// TIA Portal project "Magazzino" (V17)
// Vorlageprojekt für das Buch mit Zielsystem S7-1200

(* hardware
DEVICE "S7-1200-Station_1"  S7-1200 Station
   slot 0: "Baugruppenträger_0"  Rack  V1.0
   slot 1: "PLC_1"  CPU 1211C DC/DC/DC  6ES7 211-1AE40-0XB0  V4.1
DEVICE "HMI_1"  KTP900 Basic PN
   slot 0: "HMI_1"  KTP900 Basic PN  6AV2 123-2JB03-0AX0  17.0.0.0
   slot 1: "HMI_RT_2"  KTP900 Basic PN  6AV2 123-2JB03-0AX0  17.0.0.0
   slot 5: "HMI_1.IE_CP_1"  PROFINET Interface  17.0.0.0
      slot 1: "PROFINET Interface_1"  PROFINET Interface
         slot 1: "Port_1"  Port
*)

// ===== PLC "PLC_1"  CPU 1211C DC/DC/DC =====

VAR_GLOBAL   // PLC tag table "nastro_pacchi"
   "PaccoSens" AT %I0.0 : Bool;
   "Motor_pacchi" AT %Q0.0 : Bool;
END_VAR

VAR_GLOBAL   // PLC tag table "nastro_pedana"
   "PedanaSens" AT %I0.1 : Bool;
   "Motor_pedane" AT %Q0.1 : Bool;
END_VAR

VAR_GLOBAL   // PLC tag table "nastro_uscita"
   "FineSens" AT %I0.2 : Bool;
   "Motor" AT %Q0.2 : Bool;
END_VAR

VAR_GLOBAL   // PLC tag table "robot"
   "GoDownSens" AT %I0.3 : Bool;
   "GrabSens" AT %I0.4 : Bool;
   "MoveSens" AT %I0.5 : Bool;
   "GoDown" AT %Q0.3 : Bool;
   "Grab" AT %Q0.4 : Bool;
   "Move" AT %Q0.5 : Bool;
END_VAR

VAR_GLOBAL   // PLC tag table "allineatore"
   "AllineaSens" AT %I0.6 : Bool;
   "Allinea" AT %Q0.6 : Bool;
END_VAR

VAR_GLOBAL   // PLC tag table "bilancia"
   "BilanciaSens" AT %I1.2 : Bool;
   "Motor_bilancia" AT %Q1.1 : Bool;
   "BilanciaPeso" AT %ID30 : Real;
END_VAR

VAR_GLOBAL   // PLC tag table "stacker"
   "CentroSens" AT %I1.3 : Bool;
   "StackerMoveSens" AT %I1.4 : Bool;
   "PrelevaRSens" AT %I1.5 : Bool;
   "PrelevaLSens" AT %I1.6 : Bool;
   "AlzaSens" AT %I1.7 : Bool;
   "PrelevaR" AT %Q1.2 : Bool;
   "PrelevaL" AT %Q1.3 : Bool;
   "Alza" AT %Q1.4 : Bool;
   "Posizione" AT %QD30 : DInt;
END_VAR

VAR_GLOBAL   // PLC tag table "loader_carica"
   "CaricaSens" AT %I1.0 : Bool;
   "PaccoSuPallet" AT %I0.7 : Bool;
   "Carica" AT %Q0.7 : Bool;
END_VAR

VAR_GLOBAL   // PLC tag table "loader_scarica"
   "ScaricaSens" AT %I1.1 : Bool;
   "Scarica" AT %Q1.0 : Bool;
END_VAR

DATA_BLOCK "Database"   // DB1
{ S7_Optimized_Access := 'TRUE' }
VERSION : 0.1
   VAR
      "Mod" : Bool := true;
      Peso : Real;
      Posizione : DInt;
      CodaPesi : Array[0..4] of Real;
      HeadPesi : Int;
      TailPesi : Int;
      ArrayMagazzino : Array[0..54] of Bool;
      PosLibere : Int := 54;
   END_VAR
BEGIN
END_DATA_BLOCK

DATA_BLOCK "Magazzino_DB"   // DB2
{ S7_Optimized_Access := 'TRUE' }
VERSION : 0.1
// stored: InstanceOfName Magazzino
"Magazzino"
BEGIN
END_DATA_BLOCK

FUNCTION_BLOCK "Bilancia"   // FB1, LAD
{ S7_Optimized_Access := 'TRUE' }
VERSION : 0.1
   VAR_INPUT
      BilanciaSens : Bool;
      BilanciaPeso : Real;
      allineatore_ok : Bool;
      robot_ok : Bool;
   END_VAR
   VAR_OUTPUT
      motor_bilancia : Bool;
      p_acc : Bool;
      allineatore_start : Bool;
      robot_start : Bool;
   END_VAR
   VAR
      INIT : Bool;
      F0 : Bool;
      F1 : Bool;
      F2 : Bool;
      F3 : Bool;
      TR0 : Bool;
      TR1 : Bool;
      TR2 : Bool;
      TR3 : Bool;
      timer1 : TON_TIME;
      timer2 : TON_TIME;
      R_BilanciaSens : R_TRIG;
      F_BilanciaSens : F_TRIG;
      R_allineatore_ok : R_TRIG;
      R_F2 : R_TRIG;
      R_Inserisci : R_TRIG;
      R_robot_ok : R_TRIG;
      Inserisci : Bool;
      Salva : Bool;
   END_VAR
   VAR_TEMP   // added for the SCL form of the ladder/FBD networks
      _w1 : Bool;
   END_VAR
BEGIN

REGION Network 1: INIZIALIZZAZIONE
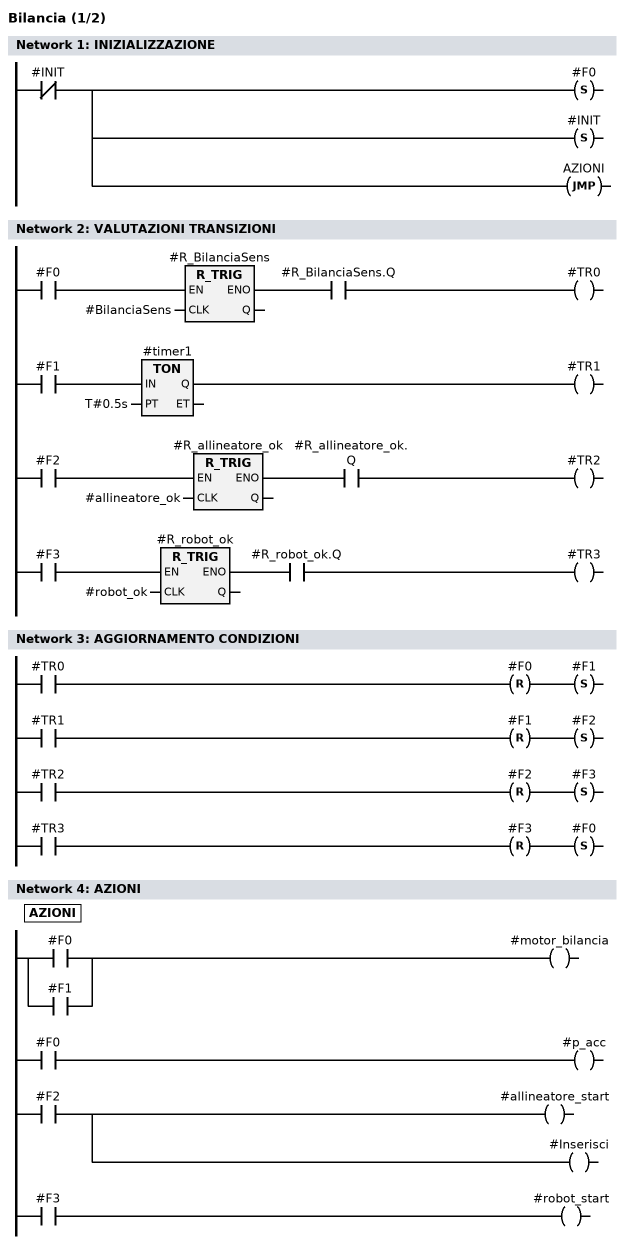
   RUNG wire#powerrail
      I_Contact( #INIT )
      wire#w1
      S_Coil( #F0 )
   END_RUNG
   RUNG wire#w1
      S_Coil( #INIT )
   END_RUNG
   RUNG wire#w1
      JumpCoil( AZIONI )
   END_RUNG
   // the same network as SCL:
   IF NOT #INIT THEN #F0 := TRUE; END_IF;
   #_w1 := NOT #INIT;
   IF #_w1 THEN
       #INIT := TRUE;
       GOTO AZIONI;
   END_IF;
END_REGION

REGION Network 2: VALUTAZIONI TRANSIZIONI
   // ENO of a box is taken as its EN; it also drops when the box reports an error
   IF #F0 THEN
       #R_BilanciaSens(CLK := #BilanciaSens);   // R_TRIG
   END_IF;
   #TR0 := #F0 AND #R_BilanciaSens.Q;
   #timer1(IN := #F1, PT := T#0.5s);   // TON
   #TR1 := #timer1.Q;
   IF #F2 THEN
       #R_allineatore_ok(CLK := #allineatore_ok);   // R_TRIG
   END_IF;
   #TR2 := #F2 AND #R_allineatore_ok.Q;
   IF #F3 THEN
       #R_robot_ok(CLK := #robot_ok);   // R_TRIG
   END_IF;
   #TR3 := #F3 AND #R_robot_ok.Q;
END_REGION

REGION Network 3: AGGIORNAMENTO CONDIZIONI
   RUNG wire#powerrail
      Contact( #TR0 )
      R_Coil( #F0 )
      S_Coil( #F1 )
   END_RUNG
   RUNG wire#powerrail
      Contact( #TR1 )
      R_Coil( #F1 )
      S_Coil( #F2 )
   END_RUNG
   RUNG wire#powerrail
      Contact( #TR2 )
      R_Coil( #F2 )
      S_Coil( #F3 )
   END_RUNG
   RUNG wire#powerrail
      Contact( #TR3 )
      R_Coil( #F3 )
      S_Coil( #F0 )
   END_RUNG
   // the same network as SCL:
   IF #TR0 THEN
       #F0 := FALSE;
       #F1 := TRUE;
   END_IF;
   IF #TR1 THEN
       #F1 := FALSE;
       #F2 := TRUE;
   END_IF;
   IF #TR2 THEN
       #F2 := FALSE;
       #F3 := TRUE;
   END_IF;
   IF #TR3 THEN
       #F3 := FALSE;
       #F0 := TRUE;
   END_IF;
END_REGION

REGION Network 4: AZIONI
   Label( AZIONI )
   RUNG wire#powerrail
      Contact( #F0 )
      wire#w1
      Coil( #motor_bilancia )
   END_RUNG
   RUNG wire#powerrail
      Contact( #F1 )
   END_RUNG wire#w1
   RUNG wire#powerrail
      Contact( #F0 )
      Coil( #p_acc )
   END_RUNG
   RUNG wire#powerrail
      Contact( #F2 )
      wire#w2
      Coil( #allineatore_start )
   END_RUNG
   RUNG wire#w2
      Coil( #Inserisci )
   END_RUNG
   RUNG wire#powerrail
      Contact( #F3 )
      Coil( #robot_start )
   END_RUNG
   // the same network as SCL:
   AZIONI:
   #motor_bilancia := #F0 OR #F1;
   #p_acc := #F0;
   #allineatore_start := #F2;
   #Inserisci := #F2;
   #robot_start := #F3;
END_REGION

REGION Network 5: GESTIONE CODA PESI
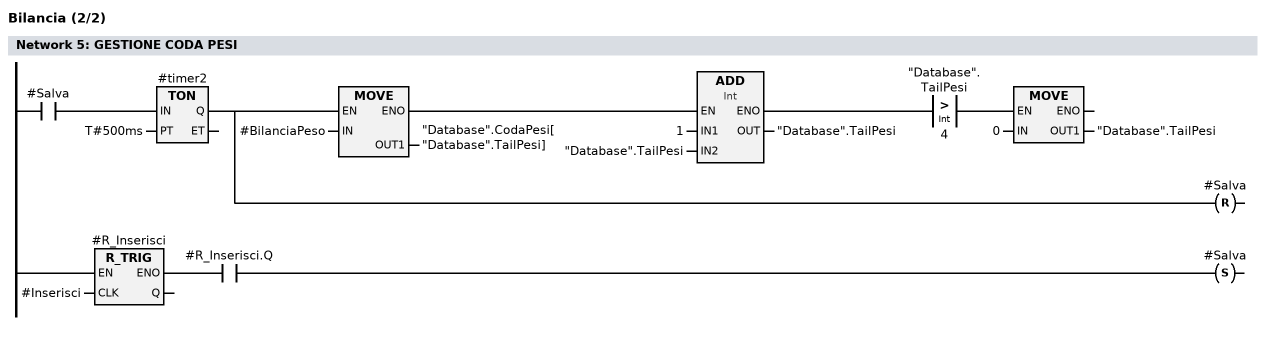
   // ENO of a box is taken as its EN; it also drops when the box reports an error
   #timer2(IN := #Salva, PT := T#500ms);   // TON
   IF #timer2.Q THEN
       "Database".CodaPesi["Database".TailPesi] := #BilanciaPeso;
       "Database".TailPesi := 1 + "Database".TailPesi;
   END_IF;
   IF #timer2.Q AND ("Database".TailPesi > 4) THEN "Database".TailPesi := 0; END_IF;
   IF #timer2.Q THEN #Salva := FALSE; END_IF;
   #R_Inserisci(CLK := #Inserisci);   // R_TRIG
   IF #R_Inserisci.Q THEN #Salva := TRUE; END_IF;
END_REGION
END_FUNCTION_BLOCK

FUNCTION_BLOCK "Robot"   // FB2, LAD
{ S7_Optimized_Access := 'TRUE' }
VERSION : 0.1
   VAR_INPUT
      MoveSens : Bool;
      GrabSens : Bool;
      GoDownSens : Bool;
      start : Bool;
      loader_ok : Bool;
   END_VAR
   VAR_OUTPUT
      Move : Bool;
      Grab : Bool;
      GoDown : Bool;
      fine : Bool;
      pacco_pronto : Bool;
   END_VAR
   VAR
      f0 : Bool;
      f1 : Bool;
      f2 : Bool;
      f3 : Bool;
      f4 : Bool;
      f5 : Bool;
      f6 : Bool;
      f7 : Bool;
      f8 : Bool;
      TR0 : Bool;
      TR1 : Bool;
      TR2 : Bool;
      TR3 : Bool;
      TR5 : Bool;
      TR6 : Bool;
      TR7 : Bool;
      TR8 : Bool;
      INIZ : Bool;
      r_prendi : R_TRIG;
      r_GrabSens : R_TRIG;
      f_GoDownSens : F_TRIG;
      f_MoveSens : F_TRIG;
      timer1 : TON_TIME;
   END_VAR
   VAR_TEMP   // added for the SCL form of the ladder/FBD networks
      _w1 : Bool;
   END_VAR
BEGIN

REGION Network 1: Inizializzazione
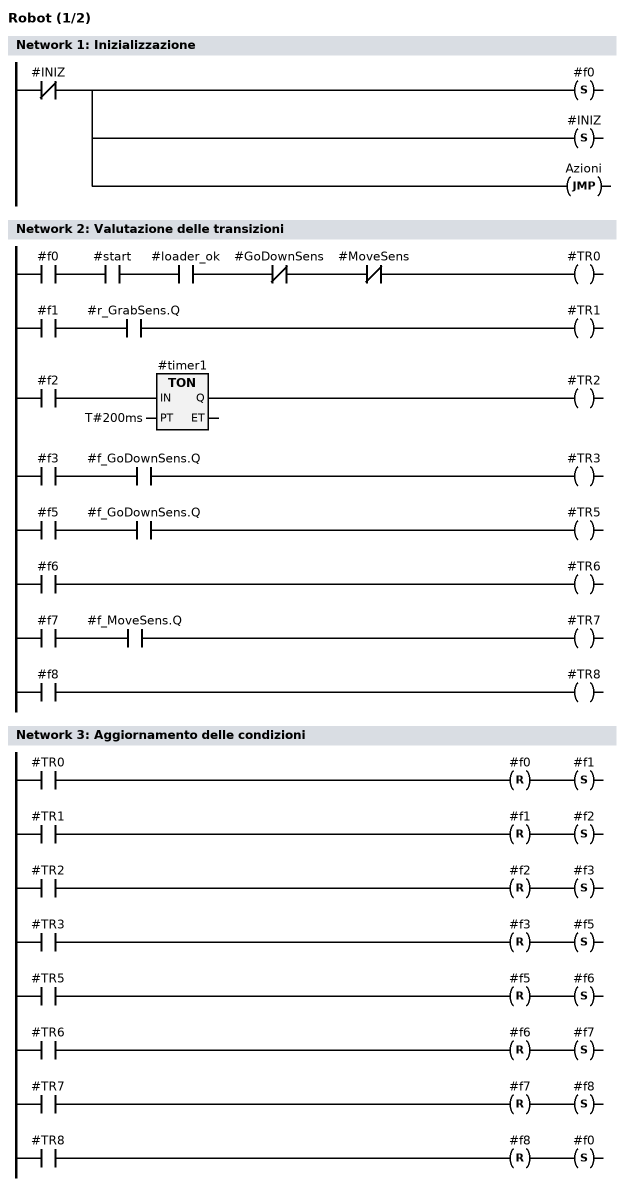
   RUNG wire#powerrail
      I_Contact( #INIZ )
      wire#w1
      S_Coil( #f0 )
   END_RUNG
   RUNG wire#w1
      S_Coil( #INIZ )
   END_RUNG
   RUNG wire#w1
      JumpCoil( Azioni )
   END_RUNG
   // the same network as SCL:
   IF NOT #INIZ THEN #f0 := TRUE; END_IF;
   #_w1 := NOT #INIZ;
   IF #_w1 THEN
       #INIZ := TRUE;
       GOTO Azioni;
   END_IF;
END_REGION

REGION Network 2: Valutazione delle transizioni
   #TR0 := #f0 AND #start AND #loader_ok AND NOT #GoDownSens AND NOT #MoveSens;
   #TR1 := #f1 AND #r_GrabSens.Q;
   #timer1(IN := #f2, PT := T#200ms);   // TON
   #TR2 := #timer1.Q;
   #TR3 := #f3 AND #f_GoDownSens.Q;
   #TR5 := #f5 AND #f_GoDownSens.Q;
   #TR6 := #f6;
   #TR7 := #f7 AND #f_MoveSens.Q;
   #TR8 := #f8;
END_REGION

REGION Network 3: Aggiornamento delle condizioni
   RUNG wire#powerrail
      Contact( #TR0 )
      R_Coil( #f0 )
      S_Coil( #f1 )
   END_RUNG
   RUNG wire#powerrail
      Contact( #TR1 )
      R_Coil( #f1 )
      S_Coil( #f2 )
   END_RUNG
   RUNG wire#powerrail
      Contact( #TR2 )
      R_Coil( #f2 )
      S_Coil( #f3 )
   END_RUNG
   RUNG wire#powerrail
      Contact( #TR3 )
      R_Coil( #f3 )
      S_Coil( #f5 )
   END_RUNG
   RUNG wire#powerrail
      Contact( #TR5 )
      R_Coil( #f5 )
      S_Coil( #f6 )
   END_RUNG
   RUNG wire#powerrail
      Contact( #TR6 )
      R_Coil( #f6 )
      S_Coil( #f7 )
   END_RUNG
   RUNG wire#powerrail
      Contact( #TR7 )
      R_Coil( #f7 )
      S_Coil( #f8 )
   END_RUNG
   RUNG wire#powerrail
      Contact( #TR8 )
      R_Coil( #f8 )
      S_Coil( #f0 )
   END_RUNG
   // the same network as SCL:
   IF #TR0 THEN
       #f0 := FALSE;
       #f1 := TRUE;
   END_IF;
   IF #TR1 THEN
       #f1 := FALSE;
       #f2 := TRUE;
   END_IF;
   IF #TR2 THEN
       #f2 := FALSE;
       #f3 := TRUE;
   END_IF;
   IF #TR3 THEN
       #f3 := FALSE;
       #f5 := TRUE;
   END_IF;
   IF #TR5 THEN
       #f5 := FALSE;
       #f6 := TRUE;
   END_IF;
   IF #TR6 THEN
       #f6 := FALSE;
       #f7 := TRUE;
   END_IF;
   IF #TR7 THEN
       #f7 := FALSE;
       #f8 := TRUE;
   END_IF;
   IF #TR8 THEN
       #f8 := FALSE;
       #f0 := TRUE;
   END_IF;
END_REGION

REGION Network 4: Azioni
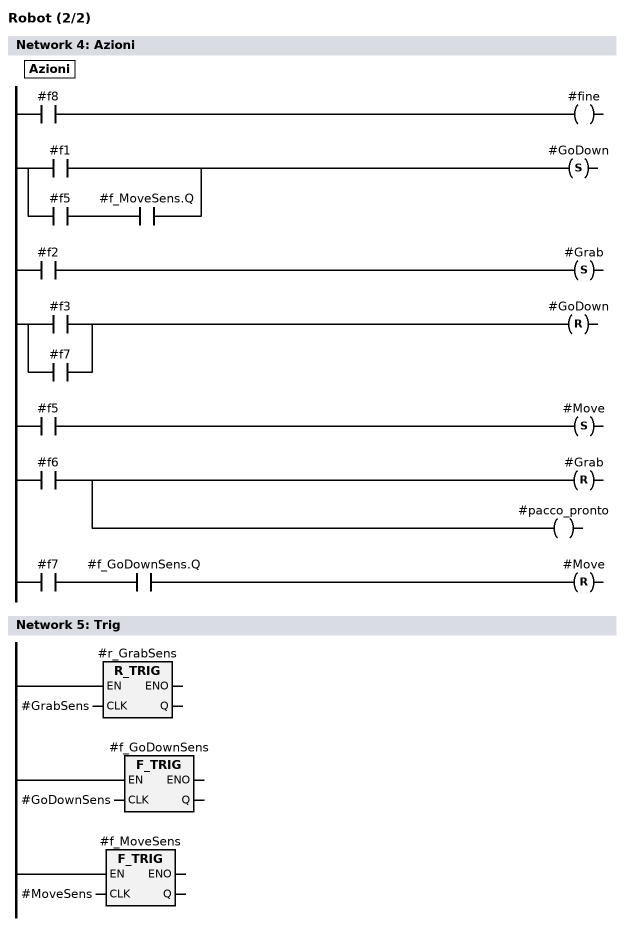
   Label( Azioni )
   RUNG wire#powerrail
      Contact( #f8 )
      Coil( #fine )
   END_RUNG
   RUNG wire#powerrail
      Contact( #f1 )
      wire#w1
      S_Coil( #GoDown )
   END_RUNG
   RUNG wire#powerrail
      Contact( #f5 )
      Contact( #f_MoveSens.Q )
   END_RUNG wire#w1
   RUNG wire#powerrail
      Contact( #f2 )
      S_Coil( #Grab )
   END_RUNG
   RUNG wire#powerrail
      Contact( #f3 )
      wire#w2
      R_Coil( #GoDown )
   END_RUNG
   RUNG wire#powerrail
      Contact( #f7 )
   END_RUNG wire#w2
   RUNG wire#powerrail
      Contact( #f5 )
      S_Coil( #Move )
   END_RUNG
   RUNG wire#powerrail
      Contact( #f6 )
      wire#w3
      R_Coil( #Grab )
   END_RUNG
   RUNG wire#w3
      Coil( #pacco_pronto )
   END_RUNG
   RUNG wire#powerrail
      Contact( #f7 )
      Contact( #f_GoDownSens.Q )
      R_Coil( #Move )
   END_RUNG
   // the same network as SCL:
   Azioni:
   #fine := #f8;
   IF #f1 OR (#f5 AND #f_MoveSens.Q) THEN #GoDown := TRUE; END_IF;
   IF #f2 THEN #Grab := TRUE; END_IF;
   IF #f3 OR #f7 THEN #GoDown := FALSE; END_IF;
   IF #f5 THEN #Move := TRUE; END_IF;
   IF #f6 THEN #Grab := FALSE; END_IF;
   #pacco_pronto := #f6;
   IF #f7 AND #f_GoDownSens.Q THEN #Move := FALSE; END_IF;
END_REGION

REGION Network 5: Trig
   #r_GrabSens(CLK := #GrabSens);   // R_TRIG
   #f_GoDownSens(CLK := #GoDownSens);   // F_TRIG
   #f_MoveSens(CLK := #MoveSens);   // F_TRIG
END_REGION
END_FUNCTION_BLOCK

FUNCTION_BLOCK "Loader"   // FB3, LAD
{ S7_Optimized_Access := 'TRUE' }
VERSION : 0.1
   VAR_INPUT
      s : Bool;
      p_dopo : Bool;
      pacco : Bool;
      flag : Bool;
   END_VAR
   VAR_OUTPUT
      motor : Bool;
      p_acc : Bool;
      posa : Bool;
      p_cons : Bool;
   END_VAR
   VAR
      INIT : Bool;
      F0 : Bool;
      F1 : Bool;
      F01 : Bool;
      F11 : Bool;
      TR0 : Bool;
      TR1 : Bool;
      TR2 : Bool;
      TR3 : Bool;
      TR4 : Bool;
      F_S : F_TRIG;
      R_S : R_TRIG;
      R_pacco : R_TRIG;
   END_VAR
   VAR_TEMP   // added for the SCL form of the ladder/FBD networks
      _w1 : Bool;
   END_VAR
BEGIN

REGION Network 1: INIZIALIZZAZIONE
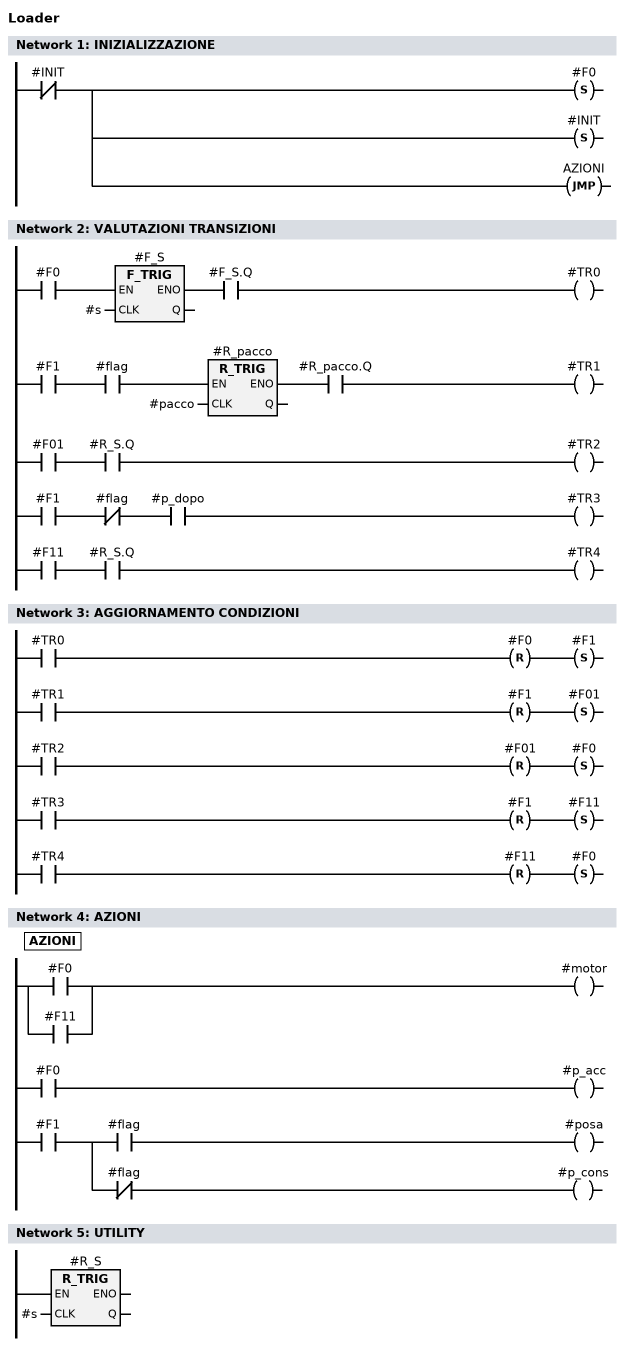
   RUNG wire#powerrail
      I_Contact( #INIT )
      wire#w1
      S_Coil( #F0 )
   END_RUNG
   RUNG wire#w1
      S_Coil( #INIT )
   END_RUNG
   RUNG wire#w1
      JumpCoil( AZIONI )
   END_RUNG
   // the same network as SCL:
   IF NOT #INIT THEN #F0 := TRUE; END_IF;
   #_w1 := NOT #INIT;
   IF #_w1 THEN
       #INIT := TRUE;
       GOTO AZIONI;
   END_IF;
END_REGION

REGION Network 2: VALUTAZIONI TRANSIZIONI
   // ENO of a box is taken as its EN; it also drops when the box reports an error
   IF #F0 THEN
       #F_S(CLK := #s);   // F_TRIG
   END_IF;
   #TR0 := #F0 AND #F_S.Q;
   #_w1 := #F1 AND #flag;
   IF #_w1 THEN
       #R_pacco(CLK := #pacco);   // R_TRIG
   END_IF;
   #TR1 := #_w1 AND #R_pacco.Q;
   #TR2 := #F01 AND #R_S.Q;
   #TR3 := #F1 AND NOT #flag AND #p_dopo;
   #TR4 := #F11 AND #R_S.Q;
END_REGION

REGION Network 3: AGGIORNAMENTO CONDIZIONI
   RUNG wire#powerrail
      Contact( #TR0 )
      R_Coil( #F0 )
      S_Coil( #F1 )
   END_RUNG
   RUNG wire#powerrail
      Contact( #TR1 )
      R_Coil( #F1 )
      S_Coil( #F01 )
   END_RUNG
   RUNG wire#powerrail
      Contact( #TR2 )
      R_Coil( #F01 )
      S_Coil( #F0 )
   END_RUNG
   RUNG wire#powerrail
      Contact( #TR3 )
      R_Coil( #F1 )
      S_Coil( #F11 )
   END_RUNG
   RUNG wire#powerrail
      Contact( #TR4 )
      R_Coil( #F11 )
      S_Coil( #F0 )
   END_RUNG
   // the same network as SCL:
   IF #TR0 THEN
       #F0 := FALSE;
       #F1 := TRUE;
   END_IF;
   IF #TR1 THEN
       #F1 := FALSE;
       #F01 := TRUE;
   END_IF;
   IF #TR2 THEN
       #F01 := FALSE;
       #F0 := TRUE;
   END_IF;
   IF #TR3 THEN
       #F1 := FALSE;
       #F11 := TRUE;
   END_IF;
   IF #TR4 THEN
       #F11 := FALSE;
       #F0 := TRUE;
   END_IF;
END_REGION

REGION Network 4: AZIONI
   Label( AZIONI )
   RUNG wire#powerrail
      Contact( #F0 )
      wire#w1
      Coil( #motor )
   END_RUNG
   RUNG wire#powerrail
      Contact( #F11 )
   END_RUNG wire#w1
   RUNG wire#powerrail
      Contact( #F0 )
      Coil( #p_acc )
   END_RUNG
   RUNG wire#powerrail
      Contact( #F1 )
      wire#w2
      Contact( #flag )
      Coil( #posa )
   END_RUNG
   RUNG wire#w2
      I_Contact( #flag )
      Coil( #p_cons )
   END_RUNG
   // the same network as SCL:
   AZIONI:
   #motor := #F0 OR #F11;
   #p_acc := #F0;
   #posa := #F1 AND #flag;
   #p_cons := #F1 AND NOT #flag;
END_REGION

REGION Network 5: UTILITY
   #R_S(CLK := #s);   // R_TRIG
END_REGION
END_FUNCTION_BLOCK

FUNCTION_BLOCK "Nastro"   // FB4, LAD
{ S7_Optimized_Access := 'TRUE' }
VERSION : 0.1
   VAR_INPUT
      s : Bool;
      p_dopo : Bool;
   END_VAR
   VAR_OUTPUT
      motor : Bool;
      p_acc : Bool;
   END_VAR
   VAR
      INIZ : Bool;
      f0 : Bool;
      f1 : Bool;
      TR0 : Bool;
      TR1 : Bool;
      f_S : F_TRIG;
      r_s : R_TRIG;
   END_VAR
   VAR_TEMP   // added for the SCL form of the ladder/FBD networks
      _w1 : Bool;
   END_VAR
BEGIN

REGION Network 1: Inizializzazione
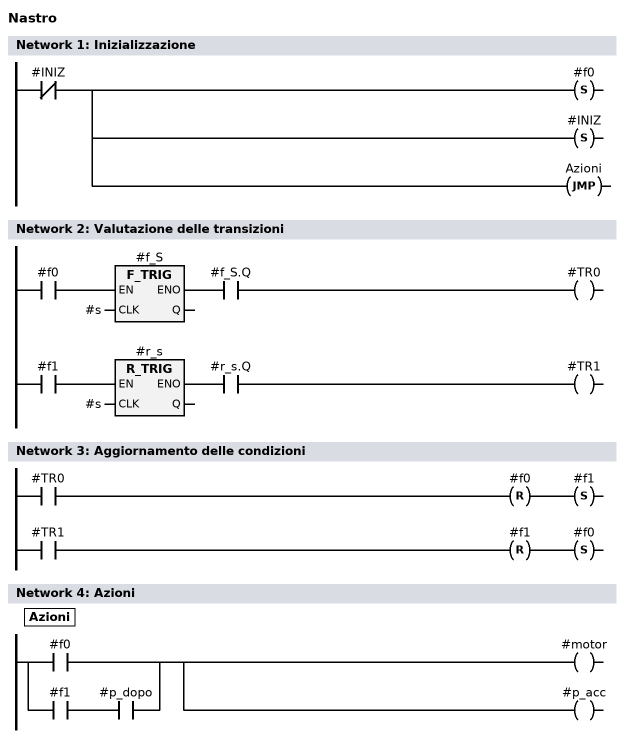
   RUNG wire#powerrail
      I_Contact( #INIZ )
      wire#w1
      S_Coil( #f0 )
   END_RUNG
   RUNG wire#w1
      S_Coil( #INIZ )
   END_RUNG
   RUNG wire#w1
      JumpCoil( Azioni )
   END_RUNG
   // the same network as SCL:
   IF NOT #INIZ THEN #f0 := TRUE; END_IF;
   #_w1 := NOT #INIZ;
   IF #_w1 THEN
       #INIZ := TRUE;
       GOTO Azioni;
   END_IF;
END_REGION

REGION Network 2: Valutazione delle transizioni
   // ENO of a box is taken as its EN; it also drops when the box reports an error
   IF #f0 THEN
       #f_S(CLK := #s);   // F_TRIG
   END_IF;
   #TR0 := #f0 AND #f_S.Q;
   IF #f1 THEN
       #r_s(CLK := #s);   // R_TRIG
   END_IF;
   #TR1 := #f1 AND #r_s.Q;
END_REGION

REGION Network 3: Aggiornamento delle condizioni
   RUNG wire#powerrail
      Contact( #TR0 )
      R_Coil( #f0 )
      S_Coil( #f1 )
   END_RUNG
   RUNG wire#powerrail
      Contact( #TR1 )
      R_Coil( #f1 )
      S_Coil( #f0 )
   END_RUNG
   // the same network as SCL:
   IF #TR0 THEN
       #f0 := FALSE;
       #f1 := TRUE;
   END_IF;
   IF #TR1 THEN
       #f1 := FALSE;
       #f0 := TRUE;
   END_IF;
END_REGION

REGION Network 4: Azioni
   Label( Azioni )
   RUNG wire#powerrail
      Contact( #f0 )
      wire#w1
      Coil( #motor )
   END_RUNG
   RUNG wire#powerrail
      Contact( #f1 )
      Contact( #p_dopo )
   END_RUNG wire#w1
   RUNG wire#w1
      Coil( #p_acc )
   END_RUNG
   // the same network as SCL:
   Azioni:
   #motor := #f0 OR (#f1 AND #p_dopo);
   #p_acc := #motor;
END_REGION
END_FUNCTION_BLOCK

FUNCTION_BLOCK "Magazzino"   // FB5, FBD
{ S7_Optimized_Access := 'TRUE' }
VERSION : 0.1
   VAR
      allineatore : "Allineatore";
      nastro_pacchi : "Nastro";
      nastro_pedane : "Nastro";
      nastro_uscita : "Nastro";
      robot : "Robot";
      loader_carica : "Loader";
      loader_scarica : "Loader";
      bilancia : "Bilancia";
      stacker : "Stacker";
   END_VAR
BEGIN

REGION Network 1
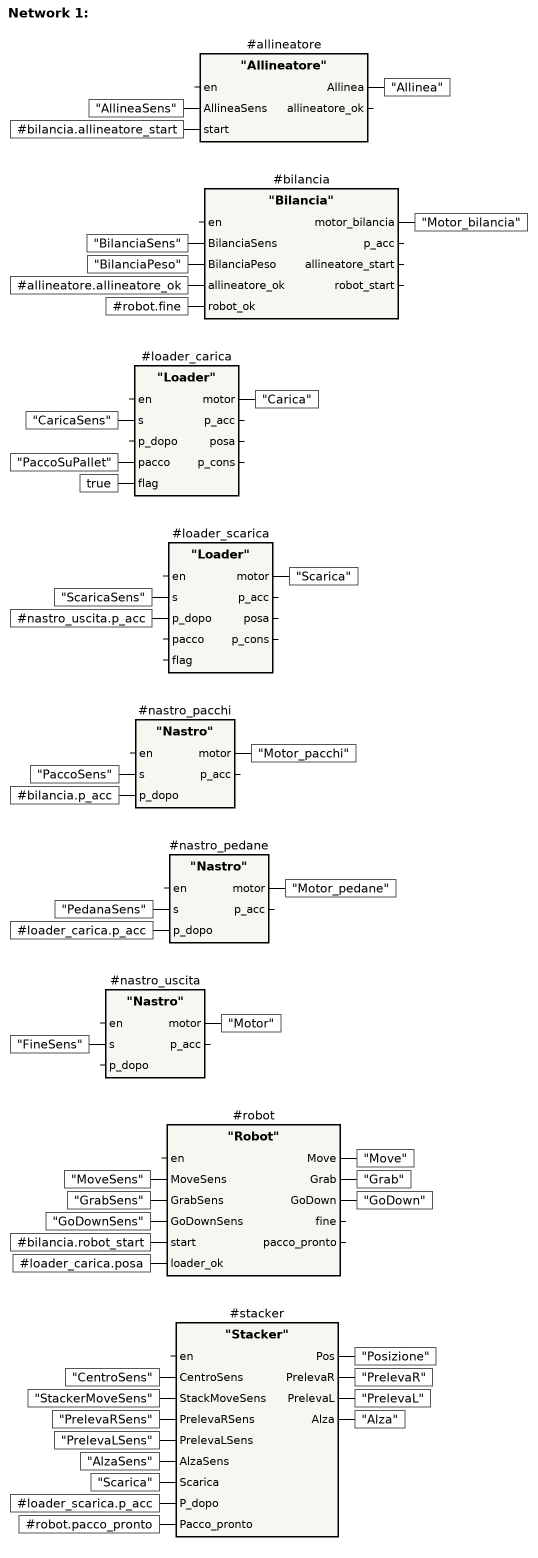
   #allineatore(AllineaSens := "AllineaSens", start := #bilancia.allineatore_start, Allinea => "Allinea");   // "Allineatore"
   #bilancia(BilanciaSens := "BilanciaSens",   // "Bilancia"
             BilanciaPeso := "BilanciaPeso",
             allineatore_ok := #allineatore.allineatore_ok,
             robot_ok := #robot.fine,
             motor_bilancia => "Motor_bilancia");
   #loader_carica(s := "CaricaSens", pacco := "PaccoSuPallet", flag := true, motor => "Carica");   // "Loader"
   #loader_scarica(s := "ScaricaSens", p_dopo := #nastro_uscita.p_acc, motor => "Scarica");   // "Loader"
   #nastro_pacchi(s := "PaccoSens", p_dopo := #bilancia.p_acc, motor => "Motor_pacchi");   // "Nastro"
   #nastro_pedane(s := "PedanaSens", p_dopo := #loader_carica.p_acc, motor => "Motor_pedane");   // "Nastro"
   #nastro_uscita(s := "FineSens", motor => "Motor");   // "Nastro"
   #robot(MoveSens := "MoveSens",   // "Robot"
          GrabSens := "GrabSens",
          GoDownSens := "GoDownSens",
          start := #bilancia.robot_start,
          loader_ok := #loader_carica.posa,
          Move => "Move",
          Grab => "Grab",
          GoDown => "GoDown");
   #stacker(CentroSens := "CentroSens",   // "Stacker"
            StackMoveSens := "StackerMoveSens",
            PrelevaRSens := "PrelevaRSens",
            PrelevaLSens := "PrelevaLSens",
            AlzaSens := "AlzaSens",
            Scarica := "Scarica",
            P_dopo := #loader_scarica.p_acc,
            Pacco_pronto := #robot.pacco_pronto,
            Pos => "Posizione",
            PrelevaR => "PrelevaR",
            PrelevaL => "PrelevaL",
            Alza => "Alza");
END_REGION
END_FUNCTION_BLOCK

FUNCTION_BLOCK "Allineatore"   // FB6, LAD
{ S7_Optimized_Access := 'TRUE' }
VERSION : 0.1
   VAR_INPUT
      AllineaSens : Bool;
      start : Bool;
   END_VAR
   VAR_OUTPUT
      Allinea : Bool;
      allineatore_ok : Bool;
   END_VAR
   VAR
      f0 : Bool;
      f1 : Bool;
      f2 : Bool;
      TR0 : Bool;
      TR1 : Bool;
      TR2 : Bool;
      INIZ : Bool;
      r_AllineaSens : R_TRIG;
      r_Start : R_TRIG;
      f_Start : F_TRIG;
   END_VAR
   VAR_TEMP   // added for the SCL form of the ladder/FBD networks
      _w1 : Bool;
   END_VAR
BEGIN

REGION Network 1: Inizializzazione
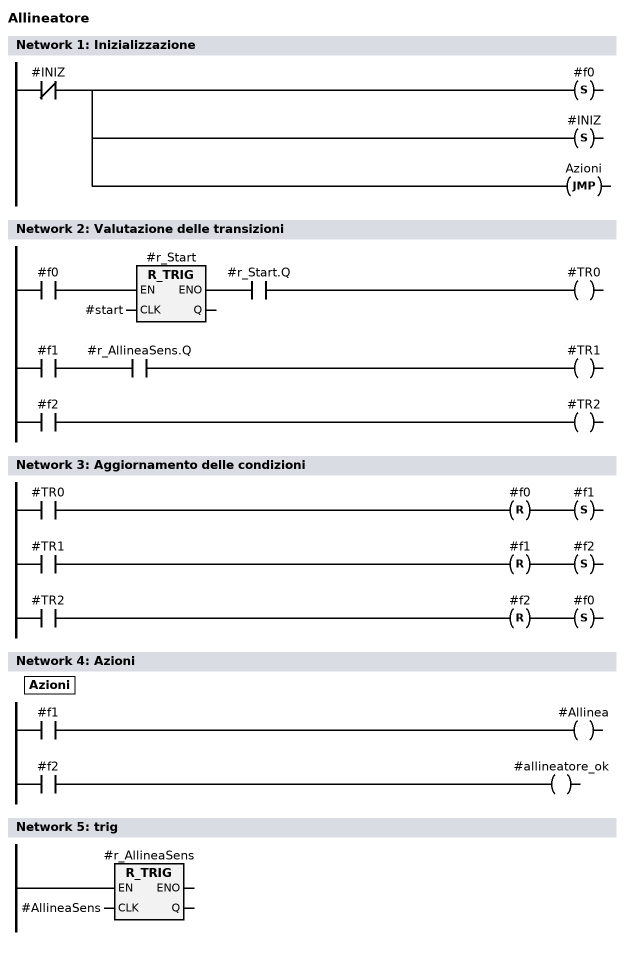
   RUNG wire#powerrail
      I_Contact( #INIZ )
      wire#w1
      S_Coil( #f0 )
   END_RUNG
   RUNG wire#w1
      S_Coil( #INIZ )
   END_RUNG
   RUNG wire#w1
      JumpCoil( Azioni )
   END_RUNG
   // the same network as SCL:
   IF NOT #INIZ THEN #f0 := TRUE; END_IF;
   #_w1 := NOT #INIZ;
   IF #_w1 THEN
       #INIZ := TRUE;
       GOTO Azioni;
   END_IF;
END_REGION

REGION Network 2: Valutazione delle transizioni
   // ENO of a box is taken as its EN; it also drops when the box reports an error
   IF #f0 THEN
       #r_Start(CLK := #start);   // R_TRIG
   END_IF;
   #TR0 := #f0 AND #r_Start.Q;
   #TR1 := #f1 AND #r_AllineaSens.Q;
   #TR2 := #f2;
END_REGION

REGION Network 3: Aggiornamento delle condizioni
   RUNG wire#powerrail
      Contact( #TR0 )
      R_Coil( #f0 )
      S_Coil( #f1 )
   END_RUNG
   RUNG wire#powerrail
      Contact( #TR1 )
      R_Coil( #f1 )
      S_Coil( #f2 )
   END_RUNG
   RUNG wire#powerrail
      Contact( #TR2 )
      R_Coil( #f2 )
      S_Coil( #f0 )
   END_RUNG
   // the same network as SCL:
   IF #TR0 THEN
       #f0 := FALSE;
       #f1 := TRUE;
   END_IF;
   IF #TR1 THEN
       #f1 := FALSE;
       #f2 := TRUE;
   END_IF;
   IF #TR2 THEN
       #f2 := FALSE;
       #f0 := TRUE;
   END_IF;
END_REGION

REGION Network 4: Azioni
   Label( Azioni )
   RUNG wire#powerrail
      Contact( #f1 )
      Coil( #Allinea )
   END_RUNG
   RUNG wire#powerrail
      Contact( #f2 )
      Coil( #allineatore_ok )
   END_RUNG
   // the same network as SCL:
   Azioni:
   #Allinea := #f1;
   #allineatore_ok := #f2;
END_REGION

REGION Network 5: trig
   #r_AllineaSens(CLK := #AllineaSens);   // R_TRIG
END_REGION
END_FUNCTION_BLOCK

FUNCTION_BLOCK "Stacker"   // FB7, LAD
{ S7_Optimized_Access := 'TRUE' }
VERSION : 0.1
   VAR_INPUT
      CentroSens : Bool;
      StackMoveSens : Bool;
      PrelevaRSens : Bool;
      PrelevaLSens : Bool;
      AlzaSens : Bool;
      Scarica : Bool;
      P_dopo : Bool;
      Pacco_pronto : Bool;
   END_VAR
   VAR_OUTPUT
      Pos : Int;
      PrelevaR : Bool;
      PrelevaL : Bool;
      Alza : Bool;
   END_VAR
   VAR
      INIT : Bool;
      F0 : Bool;
      F01 : Bool;
      F02 : Bool;
      F03 : Bool;
      F04 : Bool;
      F05 : Bool;
      F06 : Bool;
      F07 : Bool;
      F08 : Bool;
      F09 : Bool;
      F11 : Bool;
      F12 : Bool;
      F13 : Bool;
      F14 : Bool;
      F15 : Bool;
      F16 : Bool;
      F17 : Bool;
      F18 : Bool;
      R_Pacco : R_TRIG;
      F_StackMoveSens : F_TRIG;
      R_PrelevaRSens : R_TRIG;
      R_PrelevaLSens : R_TRIG;
      F_AlzaSens : F_TRIG;
      R_CentroSens : R_TRIG;
      R_F15 : R_TRIG;
      R_F14 : R_TRIG;
      F_x_ok : F_TRIG;
      F_y_ok : F_TRIG;
      R_F03 : R_TRIG;
      R_F17 : R_TRIG;
      R_F01 : R_TRIG;
      TR0 : Bool;
      TR2 : Bool;
      TR3 : Bool;
      TR4 : Bool;
      TR5 : Bool;
      TR6 : Bool;
      TR7 : Bool;
      TR8 : Bool;
      TR9 : Bool;
      TR10 : Bool;
      TR11 : Bool;
      TR12 : Bool;
      TR13 : Bool;
      TR14 : Bool;
      TR15 : Bool;
      TR16 : Bool;
      TR17 : Bool;
      TR18 : Bool;
      TR19 : Bool;
      Pacco_Presente : Bool;
      permesso : Bool;
      x_ok : Bool;
      y_ok : Bool;
   END_VAR
   VAR CONSTANT
      posIniz : Int := 21474;
   END_VAR
   VAR_TEMP   // added for the SCL form of the ladder/FBD networks
      _w1 : Bool;
      _w2 : Bool;
   END_VAR
BEGIN

REGION Network 1: INIZIALIZZAZIONE
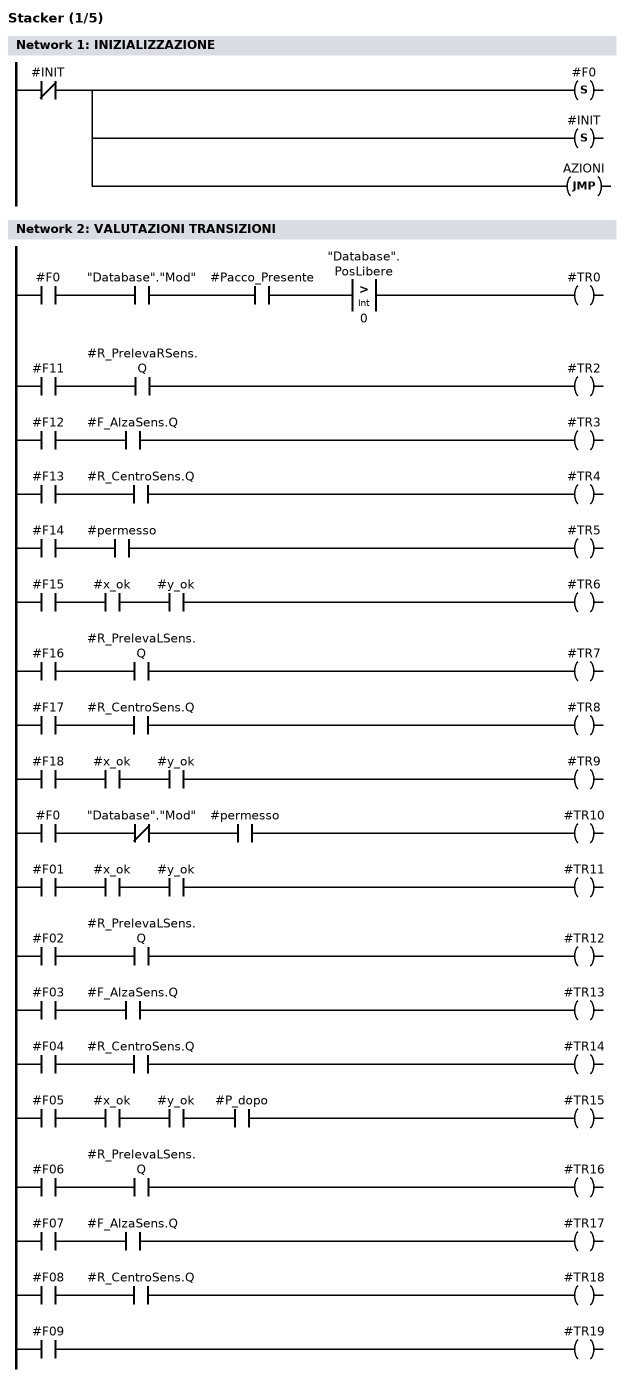
   RUNG wire#powerrail
      I_Contact( #INIT )
      wire#w1
      S_Coil( #F0 )
   END_RUNG
   RUNG wire#w1
      S_Coil( #INIT )
   END_RUNG
   RUNG wire#w1
      JumpCoil( AZIONI )
   END_RUNG
   // the same network as SCL:
   IF NOT #INIT THEN #F0 := TRUE; END_IF;
   #_w1 := NOT #INIT;
   IF #_w1 THEN
       #INIT := TRUE;
       GOTO AZIONI;
   END_IF;
END_REGION

REGION Network 2: VALUTAZIONI TRANSIZIONI
   RUNG wire#powerrail
      Contact( #F0 )
      Contact( "Database"."Mod" )
      Contact( #Pacco_Presente )
      { S7_Templates := "SrcType := Int" } GT_Contact(in1 := "Database".PosLibere, in2 := 0)
      Coil( #TR0 )
   END_RUNG
   RUNG wire#powerrail
      Contact( #F11 )
      Contact( #R_PrelevaRSens.Q )
      Coil( #TR2 )
   END_RUNG
   RUNG wire#powerrail
      Contact( #F12 )
      Contact( #F_AlzaSens.Q )
      Coil( #TR3 )
   END_RUNG
   RUNG wire#powerrail
      Contact( #F13 )
      Contact( #R_CentroSens.Q )
      Coil( #TR4 )
   END_RUNG
   RUNG wire#powerrail
      Contact( #F14 )
      Contact( #permesso )
      Coil( #TR5 )
   END_RUNG
   RUNG wire#powerrail
      Contact( #F15 )
      Contact( #x_ok )
      Contact( #y_ok )
      Coil( #TR6 )
   END_RUNG
   RUNG wire#powerrail
      Contact( #F16 )
      Contact( #R_PrelevaLSens.Q )
      Coil( #TR7 )
   END_RUNG
   RUNG wire#powerrail
      Contact( #F17 )
      Contact( #R_CentroSens.Q )
      Coil( #TR8 )
   END_RUNG
   RUNG wire#powerrail
      Contact( #F18 )
      Contact( #x_ok )
      Contact( #y_ok )
      Coil( #TR9 )
   END_RUNG
   RUNG wire#powerrail
      Contact( #F0 )
      I_Contact( "Database"."Mod" )
      Contact( #permesso )
      Coil( #TR10 )
   END_RUNG
   RUNG wire#powerrail
      Contact( #F01 )
      Contact( #x_ok )
      Contact( #y_ok )
      Coil( #TR11 )
   END_RUNG
   RUNG wire#powerrail
      Contact( #F02 )
      Contact( #R_PrelevaLSens.Q )
      Coil( #TR12 )
   END_RUNG
   RUNG wire#powerrail
      Contact( #F03 )
      Contact( #F_AlzaSens.Q )
      Coil( #TR13 )
   END_RUNG
   RUNG wire#powerrail
      Contact( #F04 )
      Contact( #R_CentroSens.Q )
      Coil( #TR14 )
   END_RUNG
   RUNG wire#powerrail
      Contact( #F05 )
      Contact( #x_ok )
      Contact( #y_ok )
      Contact( #P_dopo )
      Coil( #TR15 )
   END_RUNG
   RUNG wire#powerrail
      Contact( #F06 )
      Contact( #R_PrelevaLSens.Q )
      Coil( #TR16 )
   END_RUNG
   RUNG wire#powerrail
      Contact( #F07 )
      Contact( #F_AlzaSens.Q )
      Coil( #TR17 )
   END_RUNG
   RUNG wire#powerrail
      Contact( #F08 )
      Contact( #R_CentroSens.Q )
      Coil( #TR18 )
   END_RUNG
   RUNG wire#powerrail
      Contact( #F09 )
      Coil( #TR19 )
   END_RUNG
   // the same network as SCL:
   #TR0 := #F0 AND "Database"."Mod" AND #Pacco_Presente AND ("Database".PosLibere > 0);
   #TR2 := #F11 AND #R_PrelevaRSens.Q;
   #TR3 := #F12 AND #F_AlzaSens.Q;
   #TR4 := #F13 AND #R_CentroSens.Q;
   #TR5 := #F14 AND #permesso;
   #TR6 := #F15 AND #x_ok AND #y_ok;
   #TR7 := #F16 AND #R_PrelevaLSens.Q;
   #TR8 := #F17 AND #R_CentroSens.Q;
   #TR9 := #F18 AND #x_ok AND #y_ok;
   #TR10 := #F0 AND NOT "Database"."Mod" AND #permesso;
   #TR11 := #F01 AND #x_ok AND #y_ok;
   #TR12 := #F02 AND #R_PrelevaLSens.Q;
   #TR13 := #F03 AND #F_AlzaSens.Q;
   #TR14 := #F04 AND #R_CentroSens.Q;
   #TR15 := #F05 AND #x_ok AND #y_ok AND #P_dopo;
   #TR16 := #F06 AND #R_PrelevaLSens.Q;
   #TR17 := #F07 AND #F_AlzaSens.Q;
   #TR18 := #F08 AND #R_CentroSens.Q;
   #TR19 := #F09;
END_REGION

REGION Network 3: AGGIORNAMENTO CONDIZIONI
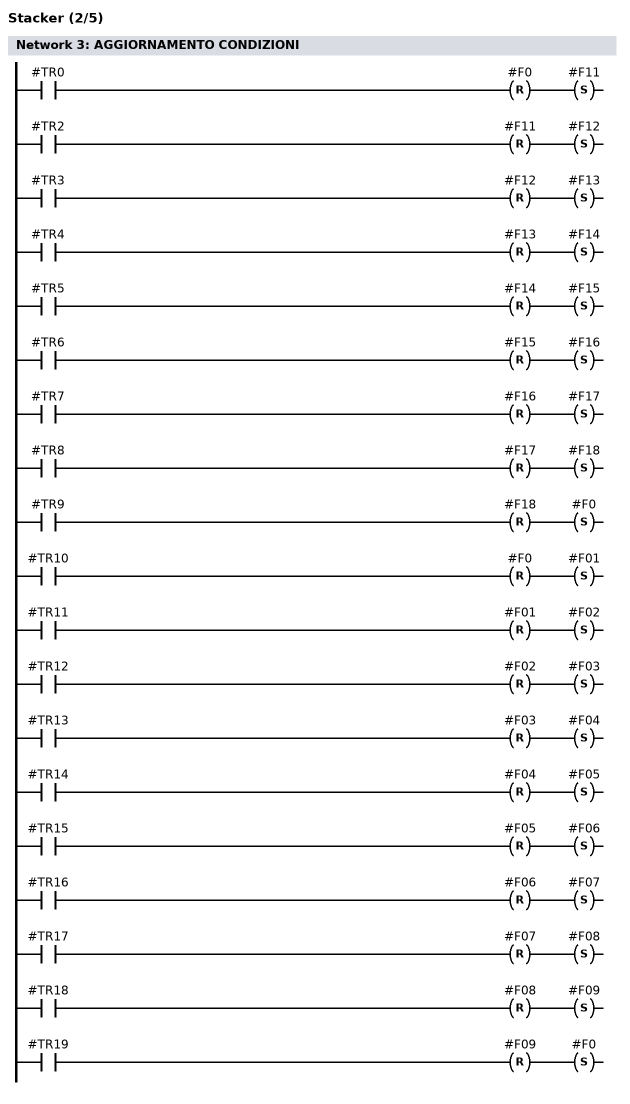
   RUNG wire#powerrail
      Contact( #TR0 )
      R_Coil( #F0 )
      S_Coil( #F11 )
   END_RUNG
   RUNG wire#powerrail
      Contact( #TR2 )
      R_Coil( #F11 )
      S_Coil( #F12 )
   END_RUNG
   RUNG wire#powerrail
      Contact( #TR3 )
      R_Coil( #F12 )
      S_Coil( #F13 )
   END_RUNG
   RUNG wire#powerrail
      Contact( #TR4 )
      R_Coil( #F13 )
      S_Coil( #F14 )
   END_RUNG
   RUNG wire#powerrail
      Contact( #TR5 )
      R_Coil( #F14 )
      S_Coil( #F15 )
   END_RUNG
   RUNG wire#powerrail
      Contact( #TR6 )
      R_Coil( #F15 )
      S_Coil( #F16 )
   END_RUNG
   RUNG wire#powerrail
      Contact( #TR7 )
      R_Coil( #F16 )
      S_Coil( #F17 )
   END_RUNG
   RUNG wire#powerrail
      Contact( #TR8 )
      R_Coil( #F17 )
      S_Coil( #F18 )
   END_RUNG
   RUNG wire#powerrail
      Contact( #TR9 )
      R_Coil( #F18 )
      S_Coil( #F0 )
   END_RUNG
   RUNG wire#powerrail
      Contact( #TR10 )
      R_Coil( #F0 )
      S_Coil( #F01 )
   END_RUNG
   RUNG wire#powerrail
      Contact( #TR11 )
      R_Coil( #F01 )
      S_Coil( #F02 )
   END_RUNG
   RUNG wire#powerrail
      Contact( #TR12 )
      R_Coil( #F02 )
      S_Coil( #F03 )
   END_RUNG
   RUNG wire#powerrail
      Contact( #TR13 )
      R_Coil( #F03 )
      S_Coil( #F04 )
   END_RUNG
   RUNG wire#powerrail
      Contact( #TR14 )
      R_Coil( #F04 )
      S_Coil( #F05 )
   END_RUNG
   RUNG wire#powerrail
      Contact( #TR15 )
      R_Coil( #F05 )
      S_Coil( #F06 )
   END_RUNG
   RUNG wire#powerrail
      Contact( #TR16 )
      R_Coil( #F06 )
      S_Coil( #F07 )
   END_RUNG
   RUNG wire#powerrail
      Contact( #TR17 )
      R_Coil( #F07 )
      S_Coil( #F08 )
   END_RUNG
   RUNG wire#powerrail
      Contact( #TR18 )
      R_Coil( #F08 )
      S_Coil( #F09 )
   END_RUNG
   RUNG wire#powerrail
      Contact( #TR19 )
      R_Coil( #F09 )
      S_Coil( #F0 )
   END_RUNG
   // the same network as SCL:
   IF #TR0 THEN
       #F0 := FALSE;
       #F11 := TRUE;
   END_IF;
   IF #TR2 THEN
       #F11 := FALSE;
       #F12 := TRUE;
   END_IF;
   IF #TR3 THEN
       #F12 := FALSE;
       #F13 := TRUE;
   END_IF;
   IF #TR4 THEN
       #F13 := FALSE;
       #F14 := TRUE;
   END_IF;
   IF #TR5 THEN
       #F14 := FALSE;
       #F15 := TRUE;
   END_IF;
   IF #TR6 THEN
       #F15 := FALSE;
       #F16 := TRUE;
   END_IF;
   IF #TR7 THEN
       #F16 := FALSE;
       #F17 := TRUE;
   END_IF;
   IF #TR8 THEN
       #F17 := FALSE;
       #F18 := TRUE;
   END_IF;
   IF #TR9 THEN
       #F18 := FALSE;
       #F0 := TRUE;
   END_IF;
   IF #TR10 THEN
       #F0 := FALSE;
       #F01 := TRUE;
   END_IF;
   IF #TR11 THEN
       #F01 := FALSE;
       #F02 := TRUE;
   END_IF;
   IF #TR12 THEN
       #F02 := FALSE;
       #F03 := TRUE;
   END_IF;
   IF #TR13 THEN
       #F03 := FALSE;
       #F04 := TRUE;
   END_IF;
   IF #TR14 THEN
       #F04 := FALSE;
       #F05 := TRUE;
   END_IF;
   IF #TR15 THEN
       #F05 := FALSE;
       #F06 := TRUE;
   END_IF;
   IF #TR16 THEN
       #F06 := FALSE;
       #F07 := TRUE;
   END_IF;
   IF #TR17 THEN
       #F07 := FALSE;
       #F08 := TRUE;
   END_IF;
   IF #TR18 THEN
       #F08 := FALSE;
       #F09 := TRUE;
   END_IF;
   IF #TR19 THEN
       #F09 := FALSE;
       #F0 := TRUE;
   END_IF;
END_REGION

REGION Network 4: AZIONI
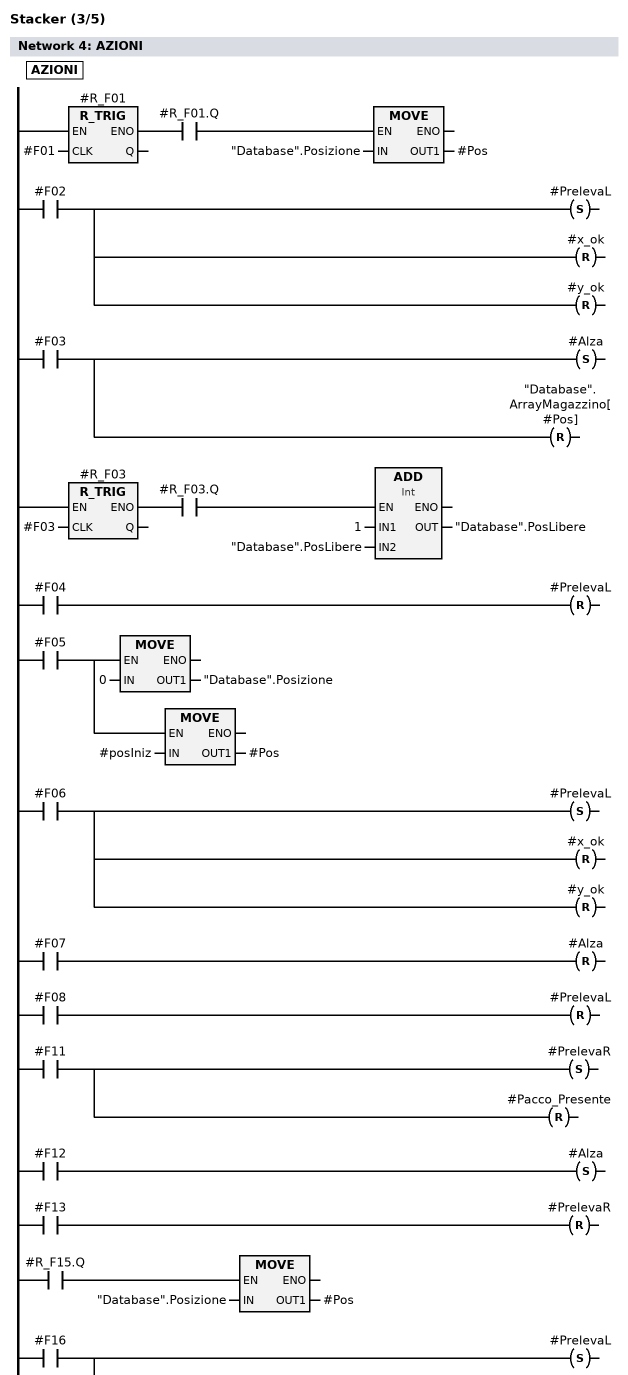
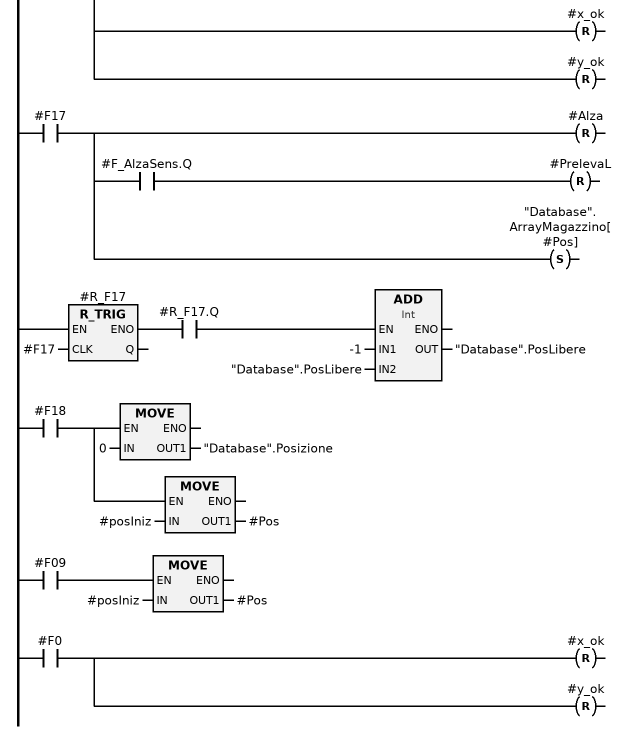
   // ENO of a box is taken as its EN; it also drops when the box reports an error
   AZIONI:
   #R_F01(CLK := #F01);   // R_TRIG
   IF #R_F01.Q THEN #Pos := "Database".Posizione; END_IF;
   IF #F02 THEN
       #PrelevaL := TRUE;
       #x_ok := FALSE;
       #y_ok := FALSE;
   END_IF;
   IF #F03 THEN
       #Alza := TRUE;
       "Database".ArrayMagazzino[#Pos] := FALSE;
   END_IF;
   #R_F03(CLK := #F03);   // R_TRIG
   IF #R_F03.Q THEN "Database".PosLibere := 1 + "Database".PosLibere; END_IF;
   IF #F04 THEN #PrelevaL := FALSE; END_IF;
   IF #F05 THEN
       "Database".Posizione := 0;
       #Pos := #posIniz;
   END_IF;
   IF #F06 THEN
       #PrelevaL := TRUE;
       #x_ok := FALSE;
       #y_ok := FALSE;
   END_IF;
   IF #F07 THEN #Alza := FALSE; END_IF;
   IF #F08 THEN #PrelevaL := FALSE; END_IF;
   IF #F11 THEN
       #PrelevaR := TRUE;
       #Pacco_Presente := FALSE;
   END_IF;
   IF #F12 THEN #Alza := TRUE; END_IF;
   IF #F13 THEN #PrelevaR := FALSE; END_IF;
   IF #R_F15.Q THEN #Pos := "Database".Posizione; END_IF;
   IF #F16 THEN
       #PrelevaL := TRUE;
       #x_ok := FALSE;
       #y_ok := FALSE;
   END_IF;
   IF #F17 THEN #Alza := FALSE; END_IF;
   IF #F17 AND #F_AlzaSens.Q THEN #PrelevaL := FALSE; END_IF;
   IF #F17 THEN "Database".ArrayMagazzino[#Pos] := TRUE; END_IF;
   #R_F17(CLK := #F17);   // R_TRIG
   IF #R_F17.Q THEN "Database".PosLibere := (-1) + "Database".PosLibere; END_IF;
   IF #F18 THEN
       "Database".Posizione := 0;
       #Pos := #posIniz;
   END_IF;
   IF #F09 THEN #Pos := #posIniz; END_IF;
   IF #F0 THEN
       #x_ok := FALSE;
       #y_ok := FALSE;
   END_IF;
END_REGION

REGION Network 5: FRONTI
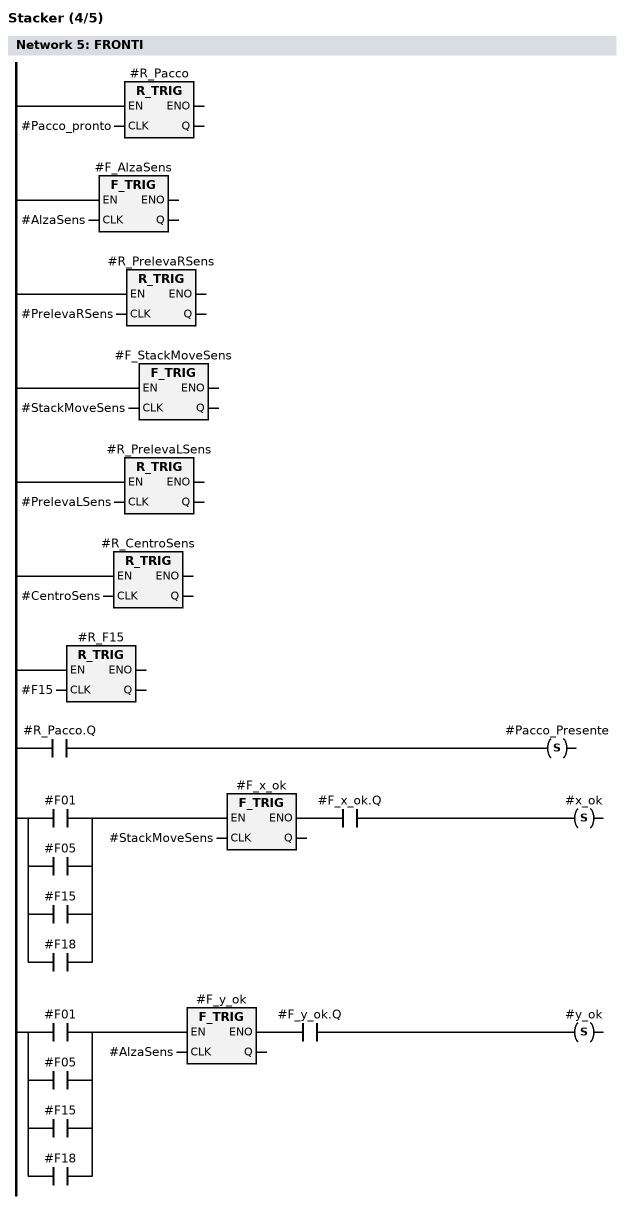
   // ENO of a box is taken as its EN; it also drops when the box reports an error
   #R_Pacco(CLK := #Pacco_pronto);   // R_TRIG
   #F_AlzaSens(CLK := #AlzaSens);   // F_TRIG
   #R_PrelevaRSens(CLK := #PrelevaRSens);   // R_TRIG
   #F_StackMoveSens(CLK := #StackMoveSens);   // F_TRIG
   #R_PrelevaLSens(CLK := #PrelevaLSens);   // R_TRIG
   #R_CentroSens(CLK := #CentroSens);   // R_TRIG
   #R_F15(CLK := #F15);   // R_TRIG
   IF #R_Pacco.Q THEN #Pacco_Presente := TRUE; END_IF;
   #_w1 := #F01 OR #F05 OR #F15 OR #F18;
   IF #_w1 THEN
       #F_x_ok(CLK := #StackMoveSens);   // F_TRIG
   END_IF;
   IF #_w1 AND #F_x_ok.Q THEN #x_ok := TRUE; END_IF;
   #_w2 := #F01 OR #F05 OR #F15 OR #F18;
   IF #_w2 THEN
       #F_y_ok(CLK := #AlzaSens);   // F_TRIG
   END_IF;
   IF #_w2 AND #F_y_ok.Q THEN #y_ok := TRUE; END_IF;
END_REGION

REGION Network 6: VALUTAZIONE PERMESSO
   // Mod = 0 -> Rimozione
   // Mod = 1 -> Inserimento
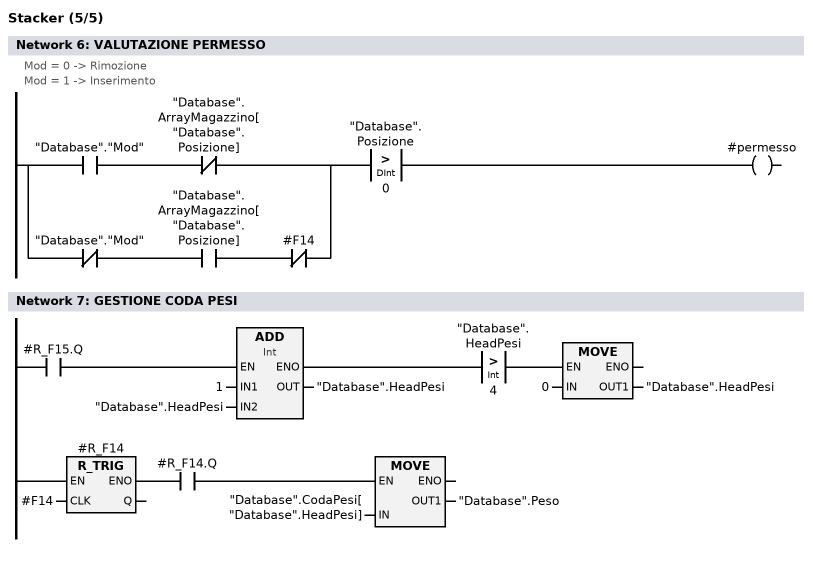
   RUNG wire#powerrail
      Contact( "Database"."Mod" )
      I_Contact( "Database".ArrayMagazzino["Database".Posizione] )
      wire#w1
      { S7_Templates := "SrcType := DInt" } GT_Contact(in1 := "Database".Posizione, in2 := 0)
      Coil( #permesso )
   END_RUNG
   RUNG wire#powerrail
      I_Contact( "Database"."Mod" )
      Contact( "Database".ArrayMagazzino["Database".Posizione] )
      I_Contact( #F14 )
   END_RUNG wire#w1
   // the same network as SCL:
   #permesso := (("Database"."Mod" AND NOT "Database".ArrayMagazzino["Database".Posizione]) OR (NOT "Database"."Mod" AND "Database".ArrayMagazzino["Database".Posizione] AND NOT #F14)) AND ("Database".Posizione > 0);
END_REGION

REGION Network 7: GESTIONE CODA PESI
   // ENO of a box is taken as its EN; it also drops when the box reports an error
   IF #R_F15.Q THEN "Database".HeadPesi := 1 + "Database".HeadPesi; END_IF;
   IF #R_F15.Q AND ("Database".HeadPesi > 4) THEN "Database".HeadPesi := 0; END_IF;
   #R_F14(CLK := #F14);   // R_TRIG
   IF #R_F14.Q THEN "Database".Peso := "Database".CodaPesi["Database".HeadPesi]; END_IF;
END_REGION
END_FUNCTION_BLOCK

FUNCTION "MHJ-PLC-Lab-Function-S71200" : Void   // FC9000, SCL
{ S7_Optimized_Access := 'TRUE' }
VERSION : 0.1
   VAR_TEMP
      rdTimeReturn : Int;
      outputTime : DTL;
      SyncVal : Byte;
      forVal : Int;
      forVal_2 : Int;
      Value : Byte;
   END_VAR
   VAR CONSTANT
      CompVal : Byte := 16#34;
      Value_01 : Byte := 16#11;
      Value_01_DW : DWord := 16#A165_D992;
      Value_02_DW : DWord := 16#58BE_4401;
   END_VAR
BEGIN

   #Value:=PEEK(area := 16#82,
        dbNumber := 0,
        byteOffset := 511);
   #Value := #Value + 1;

   POKE(area := 16#82,
        dbNumber := 0,
        byteOffset := 511,
        value := #Value);

   POKE(area:=16#81,
        dbNumber:=0,
        byteOffset:=1016,
        value:=#Value_01_DW);
   POKE(area := 16#81,
        dbNumber := 0,
        byteOffset := 1020,
        value := #Value_02_DW);

   POKE(area := 16#81,
        dbNumber := 0,
        byteOffset := 511,
        value := B#16#00);

   FOR #forVal := 0 TO 120 DO
       FOR #forVal_2:=0 TO 10 DO
           #rdTimeReturn:=RD_SYS_T(#outputTime);
           #rdTimeReturn := WR_SYS_T(#outputTime);
           #rdTimeReturn := RD_SYS_T(#outputTime);
           #rdTimeReturn := WR_SYS_T(#outputTime);
       END_FOR;
       #SyncVal:= PEEK(area := 16#81,
                      dbNumber := 0,
                      byteOffset := 511);
       IF #SyncVal = #CompVal THEN
          GOTO M_1;
       END_IF;
   END_FOR;
   RETURN;

   M_1:
   POKE(area := 16#81,
        dbNumber := 0,
        byteOffset := 511,
        value := B#16#0);
END_FUNCTION

ORGANIZATION_BLOCK "Main"   // OB1, FBD, ProgramCycle
TITLE = "Main Program Sweep (Cycle)"
{ S7_Optimized_Access := 'TRUE' }
VERSION : 0.1
   VAR_INPUT
      Initial_Call : Bool;   // Initial call of this OB
      Remanence : Bool;   // =True, if remanent data are available
   END_VAR
BEGIN

REGION Network 1: Konnektierungsbaustein für PLC-Lab
   // Im Netzwerk 1 wird der Konnektierungsbaustein für PLC-Lab aufgerufen.
   // Dieser Aufruf darf nicht entfernt werden!
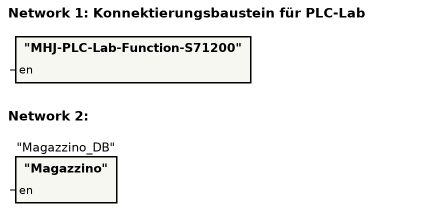
   "MHJ-PLC-Lab-Function-S71200"();
END_REGION

REGION Network 2
   "Magazzino_DB"();   // "Magazzino"
END_REGION
END_ORGANIZATION_BLOCK

(* ===== HMI "HMI_RT_2" =====
system functions are stored by id; their names below are inferred from use
connection "HMI_Connection_2": ETHERNET, SMART_S7_1200_OMS

HMI tags "Default tag table"
   "Tag_ScreenNumber" : UInt, internal
   "Posizione" : DInt = PLC Database.Posizione, 1 s
   "Pacco_Presente" : Bool = PLC Magazzino_DB.stacker.F14 AT %DB1.DBD0, 1 s
   "Mod" : Bool = PLC Database.Mod AT %DB1.DBX0.0, 1 s
   "Peso" : Real = PLC Database.Peso, 1 s
   "PosLibere" : Int = PLC Database.PosLibere AT %DB1.DBW0, 1 s

HMI tags "ArrayMagazzino"
   "Database_ArrayMagazzino{1}" : Bool = PLC Database.ArrayMagazzino[1], 1 s
   "Database_ArrayMagazzino{3}" : Bool = PLC Database.ArrayMagazzino[3], 1 s
   "Database_ArrayMagazzino{2}" : Bool = PLC Database.ArrayMagazzino[2], 1 s
   "Database_ArrayMagazzino{10}" : Bool = PLC Database.ArrayMagazzino[10], 1 s
   "Database_ArrayMagazzino{11}" : Bool = PLC Database.ArrayMagazzino[11], 1 s
   "Database_ArrayMagazzino{12}" : Bool = PLC Database.ArrayMagazzino[12], 1 s
   "Database_ArrayMagazzino{13}" : Bool = PLC Database.ArrayMagazzino[13], 1 s
   "Database_ArrayMagazzino{14}" : Bool = PLC Database.ArrayMagazzino[14], 1 s
   "Database_ArrayMagazzino{15}" : Bool = PLC Database.ArrayMagazzino[15], 1 s
   "Database_ArrayMagazzino{16}" : Bool = PLC Database.ArrayMagazzino[16], 1 s
   "Database_ArrayMagazzino{17}" : Bool = PLC Database.ArrayMagazzino[17], 1 s
   "Database_ArrayMagazzino{18}" : Bool = PLC Database.ArrayMagazzino[18], 1 s
   "Database_ArrayMagazzino{19}" : Bool = PLC Database.ArrayMagazzino[19], 1 s
   "Database_ArrayMagazzino{20}" : Bool = PLC Database.ArrayMagazzino[20], 1 s
   "Database_ArrayMagazzino{21}" : Bool = PLC Database.ArrayMagazzino[21], 1 s
   "Database_ArrayMagazzino{22}" : Bool = PLC Database.ArrayMagazzino[22], 1 s
   "Database_ArrayMagazzino{23}" : Bool = PLC Database.ArrayMagazzino[23], 1 s
   "Database_ArrayMagazzino{24}" : Bool = PLC Database.ArrayMagazzino[24], 1 s
   "Database_ArrayMagazzino{25}" : Bool = PLC Database.ArrayMagazzino[25], 1 s
   "Database_ArrayMagazzino{26}" : Bool = PLC Database.ArrayMagazzino[26], 1 s
   "Database_ArrayMagazzino{27}" : Bool = PLC Database.ArrayMagazzino[27], 1 s
   "Database_ArrayMagazzino{28}" : Bool = PLC Database.ArrayMagazzino[28], 1 s
   "Database_ArrayMagazzino{29}" : Bool = PLC Database.ArrayMagazzino[29], 1 s
   "Database_ArrayMagazzino{30}" : Bool = PLC Database.ArrayMagazzino[30], 1 s
   "Database_ArrayMagazzino{31}" : Bool = PLC Database.ArrayMagazzino[31], 1 s
   "Database_ArrayMagazzino{32}" : Bool = PLC Database.ArrayMagazzino[32], 1 s
   "Database_ArrayMagazzino{33}" : Bool = PLC Database.ArrayMagazzino[33], 1 s
   "Database_ArrayMagazzino{34}" : Bool = PLC Database.ArrayMagazzino[34], 1 s
   "Database_ArrayMagazzino{35}" : Bool = PLC Database.ArrayMagazzino[35], 1 s
   "Database_ArrayMagazzino{36}" : Bool = PLC Database.ArrayMagazzino[36], 1 s
   "Database_ArrayMagazzino{37}" : Bool = PLC Database.ArrayMagazzino[37], 1 s
   "Database_ArrayMagazzino{38}" : Bool = PLC Database.ArrayMagazzino[38], 1 s
   "Database_ArrayMagazzino{39}" : Bool = PLC Database.ArrayMagazzino[39], 1 s
   "Database_ArrayMagazzino{4}" : Bool = PLC Database.ArrayMagazzino[4], 1 s
   "Database_ArrayMagazzino{40}" : Bool = PLC Database.ArrayMagazzino[40], 1 s
   "Database_ArrayMagazzino{41}" : Bool = PLC Database.ArrayMagazzino[41], 1 s
   "Database_ArrayMagazzino{42}" : Bool = PLC Database.ArrayMagazzino[42], 1 s
   "Database_ArrayMagazzino{43}" : Bool = PLC Database.ArrayMagazzino[43], 1 s
   "Database_ArrayMagazzino{44}" : Bool = PLC Database.ArrayMagazzino[44], 1 s
   "Database_ArrayMagazzino{45}" : Bool = PLC Database.ArrayMagazzino[45], 1 s
   "Database_ArrayMagazzino{46}" : Bool = PLC Database.ArrayMagazzino[46], 1 s
   "Database_ArrayMagazzino{47}" : Bool = PLC Database.ArrayMagazzino[47], 1 s
   "Database_ArrayMagazzino{48}" : Bool = PLC Database.ArrayMagazzino[48], 1 s
   "Database_ArrayMagazzino{49}" : Bool = PLC Database.ArrayMagazzino[49], 1 s
   "Database_ArrayMagazzino{5}" : Bool = PLC Database.ArrayMagazzino[5], 1 s
   "Database_ArrayMagazzino{50}" : Bool = PLC Database.ArrayMagazzino[50], 1 s
   "Database_ArrayMagazzino{51}" : Bool = PLC Database.ArrayMagazzino[51], 1 s
   "Database_ArrayMagazzino{52}" : Bool = PLC Database.ArrayMagazzino[52], 1 s
   "Database_ArrayMagazzino{53}" : Bool = PLC Database.ArrayMagazzino[53], 1 s
   "Database_ArrayMagazzino{54}" : Bool = PLC Database.ArrayMagazzino[54], 1 s
   "Database_ArrayMagazzino{6}" : Bool = PLC Database.ArrayMagazzino[6], 1 s
   "Database_ArrayMagazzino{7}" : Bool = PLC Database.ArrayMagazzino[7], 1 s
   "Database_ArrayMagazzino{8}" : Bool = PLC Database.ArrayMagazzino[8], 1 s
   "Database_ArrayMagazzino{9}" : Bool = PLC Database.ArrayMagazzino[9], 1 s

Template "Template_1" 800x480
   Button "Exit" at 722,440 size 55x39; TextOff 'Exit'; PictureOff "ExitRuntime_KTP900_Basic_PN_TR"; PictureOn "ExitRuntime_KTP900_Basic_PN_TR"
      on Release: StopRuntime(0)
   Button "Template_Button" at 622,440 size 55x39; TextOff 'Text'
   Button "Template_Button_1" at 522,440 size 55x39; TextOff 'Text'
   Button "Template_Button_2" at 422,440 size 55x39; TextOff 'Text'
   Button "Template_Button_3" at 322,440 size 55x39; TextOff 'Text'
   Button "Template_Button_4" at 222,440 size 55x39; TextOff 'Text'
   Button "Alarms" at 122,440 size 55x39; TextOff 'Alarms'; PictureOff "AlarmDisplay_KTP900_Basic_PN_TR"; PictureOn "AlarmDisplay_KTP900_Basic_PN_TR"
      on Release: function_ef3f5d25("Alarm window_Unacknowledged", -1)
   Button "Start screen" at 22,440 size 55x39; TextOff 'Start screen'; PictureOff "NavigateHome_KTP900_Basic_PN_TR"; PictureOn "NavigateHome_KTP900_Basic_PN_TR"
      on Release: ActivateScreen("Root screen", 0)
   SymbolicIOField "Symbolic_IO_Field_Screen" at 73,7 size 620x26; TextOff '0'; TextOn '1'; TextList "TextList_ScreenNames"
      ProcessValue <- "Tag_ScreenNumber"
      on Change: ActivateScreenByNumber("Tag_ScreenNumber", 0)
   DateTimeField "HmiScreenItemData" at 695,20 size 105x20
   DateTimeField "HmiScreenItemData_1" at 695,0 size 105x20
   GraphicView "Logo" at 0,0 size 71x40; Picture "Logo of HMI_2"

screen "Root screen" 800x480, template "Template_1"
   on GenerateScreen: SetTag("Tag_ScreenNumber", 1)
   Button "Button_1" at 104,131 size 31x31; TextOff 'Text'
      on Click: SetTag("Posizione", 46)
      Appearance <- "Database_ArrayMagazzino{46}"
   Button "Button_2" at 176,131 size 31x31; TextOff 'Text'
      on Click: SetTag("Posizione", 47)
      Appearance <- "Database_ArrayMagazzino{47}"
   Button "Button_3" at 248,131 size 31x31; TextOff 'Text'
      on Click: SetTag("Posizione", 48)
      Appearance <- "Database_ArrayMagazzino{48}"
   Button "Button_4" at 320,131 size 31x31; TextOff 'Text'
      on Click: SetTag("Posizione", 49)
      Appearance <- "Database_ArrayMagazzino{49}"
   Button "Button_5" at 391,131 size 31x31; TextOff 'Text'
      on Click: SetTag("Posizione", 50)
      Appearance <- "Database_ArrayMagazzino{50}"
   Button "Button_6" at 463,131 size 31x31; TextOff 'Text'
      on Click: SetTag("Posizione", 51)
      Appearance <- "Database_ArrayMagazzino{51}"
   Button "Button_7" at 535,131 size 31x31; TextOff 'Text'
      on Click: SetTag("Posizione", 52)
      Appearance <- "Database_ArrayMagazzino{52}"
   Button "Button_8" at 607,131 size 31x31; TextOff 'Text'
      on Click: SetTag("Posizione", 53)
      Appearance <- "Database_ArrayMagazzino{53}"
   Button "Button_9" at 679,131 size 31x31; TextOff 'Text'
      on Click: SetTag("Posizione", 54)
      Appearance <- "Database_ArrayMagazzino{54}"
   Button "Button_10" at 104,183 size 31x31; TextOff 'Text'
      on Click: SetTag("Posizione", 37)
      Appearance <- "Database_ArrayMagazzino{37}"
   Button "Button_11" at 176,183 size 31x31; TextOff 'Text'
      on Click: SetTag("Posizione", 38)
      Appearance <- "Database_ArrayMagazzino{38}"
   Button "Button_12" at 248,183 size 31x31; TextOff 'Text'
      on Click: SetTag("Posizione", 39)
      Appearance <- "Database_ArrayMagazzino{39}"
   Button "Button_13" at 320,183 size 31x31; TextOff 'Text'
      on Click: SetTag("Posizione", 40)
      Appearance <- "Database_ArrayMagazzino{40}"
   Button "Button_14" at 391,183 size 31x31; TextOff 'Text'
      on Click: SetTag("Posizione", 41)
      Appearance <- "Database_ArrayMagazzino{41}"
   Button "Button_15" at 463,183 size 31x31; TextOff 'Text'
      on Click: SetTag("Posizione", 42)
      Appearance <- "Database_ArrayMagazzino{42}"
   Button "Button_16" at 535,183 size 31x31; TextOff 'Text'
      on Click: SetTag("Posizione", 43)
      Appearance <- "Database_ArrayMagazzino{43}"
   Button "Button_17" at 607,183 size 31x31; TextOff 'Text'
      on Click: SetTag("Posizione", 44)
      Appearance <- "Database_ArrayMagazzino{44}"
   Button "Button_18" at 679,183 size 31x31; TextOff 'Text'
      on Click: SetTag("Posizione", 45)
      Appearance <- "Database_ArrayMagazzino{45}"
   Button "Button_19" at 104,230 size 31x31; TextOff 'Text'
      on Click: SetTag("Posizione", 28)
      Appearance <- "Database_ArrayMagazzino{28}"
   Button "Button_20" at 176,230 size 31x31; TextOff 'Text'
      on Click: SetTag("Posizione", 29)
      Appearance <- "Database_ArrayMagazzino{29}"
   Button "Button_21" at 248,230 size 31x31; TextOff 'Text'
      on Click: SetTag("Posizione", 30)
      Appearance <- "Database_ArrayMagazzino{30}"
   Button "Button_22" at 320,230 size 31x31; TextOff 'Text'
      on Click: SetTag("Posizione", 31)
      Appearance <- "Database_ArrayMagazzino{31}"
   Button "Button_23" at 391,230 size 31x31; TextOff 'Text'
      on Click: SetTag("Posizione", 32)
      Appearance <- "Database_ArrayMagazzino{32}"
   Button "Button_24" at 463,230 size 31x31; TextOff 'Text'
      on Click: SetTag("Posizione", 33)
      Appearance <- "Database_ArrayMagazzino{33}"
   Button "Button_25" at 535,230 size 31x31; TextOff 'Text'
      on Click: SetTag("Posizione", 34)
      Appearance <- "Database_ArrayMagazzino{34}"
   Button "Button_26" at 607,230 size 31x31; TextOff 'Text'
      on Click: SetTag("Posizione", 35)
      Appearance <- "Database_ArrayMagazzino{35}"
   Button "Button_27" at 679,230 size 31x31; TextOff 'Text'
      on Click: SetTag("Posizione", 36)
      Appearance <- "Database_ArrayMagazzino{36}"
   Button "Button_28" at 105,280 size 31x31; TextOff 'Text'
      on Click: SetTag("Posizione", 19)
      Appearance <- "Database_ArrayMagazzino{19}"
   Button "Button_29" at 177,280 size 31x31; TextOff 'Text'
      on Click: SetTag("Posizione", 20)
      Appearance <- "Database_ArrayMagazzino{20}"
   Button "Button_30" at 249,280 size 31x31; TextOff 'Text'
      on Click: SetTag("Posizione", 21)
      Appearance <- "Database_ArrayMagazzino{21}"
   Button "Button_31" at 321,280 size 31x31; TextOff 'Text'
      on Click: SetTag("Posizione", 22)
      Appearance <- "Database_ArrayMagazzino{22}"
   Button "Button_32" at 392,280 size 31x31; TextOff 'Text'
      on Click: SetTag("Posizione", 23)
      Appearance <- "Database_ArrayMagazzino{23}"
   Button "Button_33" at 464,280 size 31x31; TextOff 'Text'
      on Click: SetTag("Posizione", 24)
      Appearance <- "Database_ArrayMagazzino{24}"
   Button "Button_34" at 536,280 size 31x31; TextOff 'Text'
      on Click: SetTag("Posizione", 25)
      Appearance <- "Database_ArrayMagazzino{25}"
   Button "Button_35" at 608,280 size 31x31; TextOff 'Text'
      on Click: SetTag("Posizione", 26)
      Appearance <- "Database_ArrayMagazzino{26}"
   Button "Button_36" at 680,280 size 31x31; TextOff 'Text'
      on Click: SetTag("Posizione", 27)
      Appearance <- "Database_ArrayMagazzino{27}"
   Button "Button_37" at 104,325 size 31x31; TextOff 'Text'
      on Click: SetTag("Posizione", 10)
      Appearance <- "Database_ArrayMagazzino{10}"
   Button "Button_38" at 176,325 size 31x31; TextOff 'Text'
      on Click: SetTag("Posizione", 11)
      Appearance <- "Database_ArrayMagazzino{11}"
   Button "Button_39" at 248,325 size 31x31; TextOff 'Text'
      on Click: SetTag("Posizione", 12)
      Appearance <- "Database_ArrayMagazzino{12}"
   Button "Button_40" at 320,325 size 31x31; TextOff 'Text'
      on Click: SetTag("Posizione", 13)
      Appearance <- "Database_ArrayMagazzino{13}"
   Button "Button_41" at 391,325 size 31x31; TextOff 'Text'
      on Click: SetTag("Posizione", 14)
      Appearance <- "Database_ArrayMagazzino{14}"
   Button "Button_42" at 463,325 size 31x31; TextOff 'Text'
      on Click: SetTag("Posizione", 15)
      Appearance <- "Database_ArrayMagazzino{15}"
   Button "Button_43" at 535,325 size 31x31; TextOff 'Text'
      on Click: SetTag("Posizione", 16)
      Appearance <- "Database_ArrayMagazzino{16}"
   Button "Button_44" at 607,325 size 31x31; TextOff 'Text'
      on Click: SetTag("Posizione", 17)
      Appearance <- "Database_ArrayMagazzino{17}"
   Button "Button_45" at 679,325 size 31x31; TextOff 'Text'
      on Click: SetTag("Posizione", 18)
      Appearance <- "Database_ArrayMagazzino{18}"
   Button "Button_46" at 104,372 size 31x31; TextOff 'Text'
      on Click: SetTag("Posizione", 1)
      Appearance <- "Database_ArrayMagazzino{1}"
   Button "Button_47" at 176,372 size 31x31; TextOff 'Text'
      on Click: SetTag("Posizione", 2)
      Appearance <- "Database_ArrayMagazzino{2}"
   Button "Button_48" at 248,372 size 31x31; TextOff 'Text'
      on Click: SetTag("Posizione", 3)
      Appearance <- "Database_ArrayMagazzino{3}"
   Button "Button_49" at 320,372 size 31x31; TextOff 'Text'
      on Click: SetTag("Posizione", 4)
      Appearance <- "Database_ArrayMagazzino{4}"
   Button "Button_50" at 391,372 size 31x31; TextOff 'Text'
      on Click: SetTag("Posizione", 5)
      Appearance <- "Database_ArrayMagazzino{5}"
   Button "Button_51" at 463,372 size 31x31; TextOff 'Text'
      on Click: SetTag("Posizione", 6)
      Appearance <- "Database_ArrayMagazzino{6}"
   Button "Button_52" at 535,372 size 31x31; TextOff 'Text'
      on Click: SetTag("Posizione", 7)
      Appearance <- "Database_ArrayMagazzino{7}"
   Button "Button_53" at 607,372 size 31x31; TextOff 'Text'
      on Click: SetTag("Posizione", 8)
      Appearance <- "Database_ArrayMagazzino{8}"
   Button "Button_54" at 679,372 size 31x31; TextOff 'Text'
      on Click: SetTag("Posizione", 9)
      Appearance <- "Database_ArrayMagazzino{9}"
   TextField "Text field_2" at 61,371 size 18x32; Text '1'
   TextField "Text field_3" at 59,325 size 18x32; Text '2'
   TextField "Text field_4" at 60,280 size 18x32; Text '3'
   TextField "Text field_5" at 61,229 size 18x32; Text '4'
   TextField "Text field_6" at 61,183 size 18x32; Text '5'
   TextField "Text field_7" at 60,132 size 18x32; Text '6'
   TextField "Text field_8" at 110,89 size 18x32; Text '1'
   TextField "Text field_9" at 183,89 size 18x32; Text '2'
   TextField "Text field_10" at 256,89 size 18x32; Text '3'
   TextField "Text field_11" at 325,89 size 18x32; Text '4'
   TextField "Text field_12" at 396,89 size 18x32; Text '5'
   TextField "Text field_13" at 469,89 size 18x32; Text '6'
   TextField "Text field_14" at 542,89 size 18x32; Text '7'
   TextField "Text field_15" at 611,89 size 18x32; Text '8'
   TextField "Text field_16" at 684,89 size 18x32; Text '9'
   TextField "Text field_1" at 201,42 size 213x41; Text 'Pacco pronto'
      Appearance <- "Pacco_Presente"
      Visibility <- "Pacco_Presente"
   Switch "Switch_1" at 662,44 size 111x38; TextOn 'CARICA'; CaptionText 'Switch'; TextOff 'SCARICA'
      ProcessValue <- "Mod"
   IOField "I/O field_1" at 533,49 size 96x32; FormatPattern 99.99
      Visibility <- "Pacco_Presente"
      ProcessValue <- "Peso"
   TextField "Text field_17" at 438,49 size 71x34; Text 'PESO'
      Visibility <- "Pacco_Presente"
   IOField "I/O field_2" at 14,51 size 96x32; FormatPattern 99
      ProcessValue <- "PosLibere"
*)